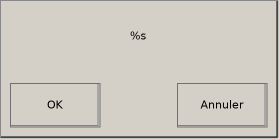
VISUALIZATION UTIL_CONFIRM  // 279x139
VAR_INPUT
	Num_Text:		INT;
END_VAR
VAR_IN_OUT
	OrdreDD:		BOOL;
	Visu:			BOOL;	
END_VAR
    RoundedRectangle (0,0 277x137)
    Textfield (19,6 238x60), "%s", text list: 'TextList_Users_Menu', text index: Num_Text
    Button (10,83 90x44), "OK"
        OnMouseClick: execute { OrdreDD:=(TRUE); }
        OnMouseClick: execute { Visu:=(FALSE); }
    Button (177,83 90x44), "Annuler"
        OnMouseClick: execute { Visu:=(FALSE); }
END_VISUALIZATION

(* stored: Version 1.1.0.1, ProductVersion 3.1.4024.10
   Visu UTIL_CONFIRM: Id {a93f950e-c9ef-4742-963a-800e2b1b080f} *)
